# B&R Automation Studio project A2019059_Linka_Power_CP (part 29)

```iecst
        273:
            SC_P2_Srobovanie.StepName:='273 - Automaticky Rezim - model 5F, zasunutie skrutkovacky M4 a vypnutie prisavania skrutky';
            SC_P2_Srobovanie.IdleTime.PT:= T#200ms;
            SC_P2_Srobovanie.AlarmTime.PT:= T#5s;

            IF NOT SC_P2_Srobovanie.Switch1 THEN
                P2_Srobovanie.OUT.SkrutkM4_VYSUN_YV24:= FALSE;
                P2_Srobovanie.OUT.SkrutkM4_PrisavSkrutky_RUN_YV26:= FALSE;
                SC_P2_Srobovanie.Switch1:= TRUE;
            END_IF

            IF P2_Srobovanie.IN.SkrutkM4_ZASUNUTY_MS10 THEN
                SC_P2_Srobovanie.ResetStep:= TRUE;
                SC_P2_Srobovanie.Step:= 274;
            END_IF

        274:
            SC_P2_Srobovanie.StepName:='274 - Automaticky Rezim - model 5F, signal skrutka M4 odobrata';
            SC_P2_Srobovanie.IdleTime.PT:= T#200ms;
            SC_P2_Srobovanie.AlarmTime.PT:= T#5s;

            IF NOT SC_P2_Srobovanie.Switch1 THEN
                P2_Srobovanie.SkrutkovaciSet_M4.SkrutkaM4_Odobrata:= TRUE;
                SC_P2_Srobovanie.Switch1:= TRUE;
            END_IF

            IF NOT P2_Srobovanie.SkrutkovaciSet_M4.SkrutkaM4_Pripravena THEN
                P2_Srobovanie.SkrutkovaciSet_M4.SkrutkaM4_Odobrata:= FALSE;
                SC_P2_Srobovanie.ResetStep:= TRUE;
                SC_P2_Srobovanie.Step:= 275;
            END_IF

        275:
            SC_P2_Srobovanie.StepName:='275 - Automaticky Rezim - model 5F, kontrola vysledkov skrutkovania pravej skrutky M4';
            SC_P2_Srobovanie.IdleTime.PT:= T#200ms;
            SC_P2_Srobovanie.AlarmTime.PT:= T#5s;

            IF P2_Srobovanie.Skrutkovacka_M4.Stav_VysledokUtahovania_OK THEN
                P2_Srobovanie.STAV.Vysledok_Srobovania:= 'OK';
                P2_Srobovanie.OUT.KOM_Srobovanie_Ukoncene:= TRUE;
                SC_P2_Srobovanie.ResetStep:= TRUE;
                SC_P2_Srobovanie.Step:= 278;
            ELSIF P2_Srobovanie.Skrutkovacka_M4.Stav_VysledokUtahovania_NG THEN
                P2_Srobovanie.STAV.Vysledok_Srobovania:= 'NG';
                P2_Srobovanie.OUT.KOM_Srobovanie_Ukoncene:= TRUE;
                SC_P2_Srobovanie.ResetStep:= TRUE;
                SC_P2_Srobovanie.Step:= 278;
            END_IF

        278:
            SC_P2_Srobovanie.StepName:='278 - Automaticky Rezim - model 5F, cakam na zrusenie signalu zaskrutkuj pravu srobu M4';
            SC_P2_Srobovanie.IdleTime.PT:= T#200ms;
            SC_P2_Srobovanie.AlarmTime.PT:= T#5s;

            IF NOT P2_StoperSrobovania.OUT.KOM_5F_ZasrobujPravuSkrutkuM4 THEN
                P2_Srobovanie.OUT.KOM_Srobovanie_Ukoncene:= FALSE;
                SC_P2_Srobovanie.ResetStep:= TRUE;
                SC_P2_Srobovanie.Step:= 100;
            END_IF

            //**********************************************************************Model 5H*******************************************************************************************//
            //Zaskrutkovanie lavej skrutky M5//

        300:
            SC_P2_Srobovanie.StepName:='300 - Automaticky Rezim - model 5H, napolohovanie zadnej skrutkovacky M5 na poziciu lavej skrutky M5';
            SC_P2_Srobovanie.IdleTime.PT:= T#200ms;
            SC_P2_Srobovanie.AlarmTime.PT:= T#5s;

            P2_Robot.KOM_OUT.ManipSrobovania_BezpecnaPozicia:= FALSE;

            P2_Srobovanie.PAR.OsX_ZadanaPozicia:= P2_RemPremenne.P2_Srob5H_PozX_LavejSkrutkyM5; //mm
            P2_Srobovanie.PAR.OsY_ZadanaPozicia:= P2_RemPremenne.P2_Srob5H_PozY_LavejSkrutkyM5; //mm

            IF NOT SC_P2_Srobovanie.Switch1 AND SC_OvlManipulatora_OsX.Step = 1 AND SC_OvlManipulatora_OsY.Step = 1 AND P2_Srobovacky_VychodziaPozicia AND Safety.STAV.P2_ZonaBunky_AKTIVNA  THEN
                OsX_POLOHUJ:= TRUE;
                OsY_POLOHUJ:= TRUE;
                SC_P2_Srobovanie.Switch1:= TRUE;
            END_IF

            IF P2_Srobovanie.STAV.OsX_PoziciaDosiahnuta AND P2_Srobovanie.STAV.OsY_PoziciaDosiahnuta THEN
                P2_Srobovanie.STAV.OsX_PoziciaDosiahnuta:= FALSE;
                P2_Srobovanie.STAV.OsY_PoziciaDosiahnuta:= FALSE;
                IF P2_Srobovanie.RR_PolohujNaPoziciuSkrutky_5H THEN
                    P2_Srobovanie.RR_PolohujNaPoziciuSkrutky_5H:= FALSE;
                    P2_Srobovanie.RR_PolohujNaPoziciuSkrutky_4F:= FALSE;
                    P2_Srobovanie.RR_PolohujNaPoziciuSkrutky_5F:= FALSE;
                    SC_P2_Srobovanie.ResetStep:= TRUE;
                    SC_P2_Srobovanie.Step:= 700;
                ELSE
                    SC_P2_Srobovanie.ResetStep:= TRUE;
                    SC_P2_Srobovanie.Step:= 303;
                END_IF
            END_IF

        303:
            SC_P2_Srobovanie.StepName:='303 - Automaticky Rezim - model 5H, vymazanie vysledkov srobovania';
            SC_P2_Srobovanie.IdleTime.PT:= T#2s;
            SC_P2_Srobovanie.AlarmTime.PT:= T#5s;

            IF NOT SC_P2_Srobovanie.Switch1 THEN
                P2_Srobovanie.Skrutkovacka_M5.RESET_Vysledkov:= TRUE;
                SC_P2_Srobovanie.Switch1:= TRUE;
            END_IF

            IF NOT P2_Srobovanie.Skrutkovacka_M5.Stav_VysledokUtahovania_NG AND NOT P2_Srobovanie.Skrutkovacka_M5.Stav_VysledokUtahovania_OK AND NOT P2_Srobovanie.Skrutkovacka_M5.Stav_UtahovanieUkoncene THEN
                P2_Srobovanie.Skrutkovacka_M5.RESET_Vysledkov:= FALSE;
                SC_P2_Srobovanie.ResetStep:= TRUE;
                SC_P2_Srobovanie.Step:= 305;
            END_IF

        305:
            SC_P2_Srobovanie.StepName:='305 - Automaticky Rezim - model 5H, kontrola skrutky M5 v skrutkovacke';
            SC_P2_Srobovanie.IdleTime.PT:= T#5s;
            SC_P2_Srobovanie.AlarmTime.PT:= T#30s;
            SC_P2_Srobovanie.AlarmTime.IN:= TRUE;

            IF P2_Srobovanie.SkrutkovaciSet_M5.SkrutkaM5_Pripravena AND P2_Srobovanie.Skrutkovacka_M5.Stav_READY_to_START AND NOT PAUZA THEN
                SC_P2_Srobovanie.ResetStep:= TRUE;
                SC_P2_Srobovanie.Step:= 308;
            ELSIF SC_P2_Srobovanie.AlarmTime.Q THEN
                IF NOT P2_Srobovanie.SkrutkovaciSet_M5.SkrutkaM5_Pripravena THEN
                    P2_Alarmy[238]:= TRUE;
                END_IF
                IF NOT P2_Srobovanie.Skrutkovacka_M5.Stav_READY_to_START THEN
                    P2_Alarmy[276]:= TRUE;
                END_IF
                P2_StoperSrobovania.STAV.Porucha:= TRUE;
                P2_Srobovanie.OUT.KOM_Srobovanie_Ukoncene:= TRUE;
                SC_P2_Srobovanie.ResetStep:= TRUE;
                SC_P2_Srobovanie.Step:= 318;
            END_IF

        308:
            SC_P2_Srobovanie.StepName:='308 - Automaticky Rezim - model 5H, vysunutie skrutkovacky M5';
            SC_P2_Srobovanie.IdleTime.PT:= T#2s;
            SC_P2_Srobovanie.AlarmTime.PT:= T#5s;

            SC_P2_Srobovanie.AlarmTime.IN:= (P2_Srobovanie.IN.SkrutkM5_VysunutieHrotu_IOS5 < 2);

            IF NOT SC_P2_Srobovanie.Switch1 THEN
                P2_Srobovanie.OUT.SkrutkM5_PrisavSkrutky_RUN_YV16:= TRUE;
                P2_Srobovanie.OUT.SkrutkM5_VYSUN_YV14:= TRUE;
                P2_Srobovanie.Skrutkovacka_M5.START_Utahovania:= TRUE;
                SC_P2_Srobovanie.Switch1:= TRUE;
            END_IF

            IF NOT P2_Srobovanie.Skrutkovacka_M5.Stav_UtahovanieUkoncene AND P2_Srobovanie.IN.SkrutkM5_VysunutieHrotu_IOS5 > 2 AND NOT TEST THEN
                SC_P2_Srobovanie.ResetStep:= TRUE;
                SC_P2_Srobovanie.Step:= 310;
            ELSIF SC_P2_Srobovanie.AlarmTime.Q AND NOT TEST THEN
                P2_Alarmy[269]:= TRUE;
                P2_StoperSrobovania.STAV.Porucha:= TRUE;
                P2_Srobovanie.OUT.SkrutkM5_VYSUN_YV14:= FALSE;
                P2_Srobovanie.Skrutkovacka_M5.START_Utahovania:= FALSE;
                P2_Srobovanie.OUT.KOM_Srobovanie_Ukoncene:= TRUE;
                SC_P2_Srobovanie.ResetStep:= TRUE;
                SC_P2_Srobovanie.Step:= 318;
            END_IF

        310:
            SC_P2_Srobovanie.StepName:='310 - Automaticky Rezim - model 5H, cakam na ukoncenie skrutkovania skrutkovacky M5';
            SC_P2_Srobovanie.IdleTime.PT:= T#30s;
            SC_P2_Srobovanie.AlarmTime.PT:= T#10s;
            SC_P2_Srobovanie.IdleTime.IN:= TRUE;
            SC_P2_Srobovanie.AlarmTime.IN:= TRUE;

            IF P2_Srobovanie.Skrutkovacka_M5.Stav_UtahovanieUkoncene THEN
                P2_Srobovanie.Skrutkovacka_M5.START_Utahovania:= FALSE;
                CasSrobovania:= TIME_TO_REAL(SC_P2_Srobovanie.IdleTime.ET);
                Reports.Skrutkovacky.VyskaSkrutkovania.P2_LavaSkrutkaM5:= REAL_TO_STRING(P2_Srobovanie.IN.SkrutkM5_VysunutieHrotu_IOS5);
                Reports.Skrutkovacky.CasSkrutkovania.P2_LavaSkrutkaM5:= REAL_TO_STRING(CasSrobovania/1000);
                SC_P2_Srobovanie.ResetStep:= TRUE;
                SC_P2_Srobovanie.Step:= 313;
            ELSIF SC_P2_Srobovanie.AlarmTime.Q THEN
                P2_Alarmy[273]:= TRUE;
                P2_StoperSrobovania.STAV.Porucha:= TRUE;
                P2_Srobovanie.OUT.SkrutkM5_VYSUN_YV14:= FALSE;
                P2_Srobovanie.Skrutkovacka_M5.START_Utahovania:= FALSE;
                P2_Srobovanie.OUT.KOM_Srobovanie_Ukoncene:= TRUE;
                SC_P2_Srobovanie.ResetStep:= TRUE;
                SC_P2_Srobovanie.Step:= 318;
            END_IF

        313:
            SC_P2_Srobovanie.StepName:='313 - Automaticky Rezim - model 5H, zasunutie skrutkovacky M5 a vypnutie prisavania skrutky';
            SC_P2_Srobovanie.IdleTime.PT:= T#200ms;
            SC_P2_Srobovanie.AlarmTime.PT:= T#5s;

            IF NOT SC_P2_Srobovanie.Switch1 THEN
                P2_Srobovanie.OUT.SkrutkM5_VYSUN_YV14:= FALSE;
                P2_Srobovanie.OUT.SkrutkM5_PrisavSkrutky_RUN_YV16:= FALSE;
                SC_P2_Srobovanie.Switch1:= TRUE;
            END_IF

            IF P2_Srobovanie.IN.SkrutkM5_ZASUNUTY_MS11 THEN
                SC_P2_Srobovanie.ResetStep:= TRUE;
                SC_P2_Srobovanie.Step:= 314;
            END_IF

        314:
            SC_P2_Srobovanie.StepName:='314 - Automaticky Rezim - model 5H, signal skrutka M5 odobrata';
            SC_P2_Srobovanie.IdleTime.PT:= T#200ms;
            SC_P2_Srobovanie.AlarmTime.PT:= T#5s;

            IF NOT SC_P2_Srobovanie.Switch1 THEN
                P2_Srobovanie.SkrutkovaciSet_M5.SkrutkaM5_Odobrata:= TRUE;
                SC_P2_Srobovanie.Switch1:= TRUE;
            END_IF

            IF NOT P2_Srobovanie.SkrutkovaciSet_M5.SkrutkaM5_Pripravena THEN
                P2_Srobovanie.SkrutkovaciSet_M5.SkrutkaM5_Odobrata:= FALSE;
                SC_P2_Srobovanie.ResetStep:= TRUE;
                SC_P2_Srobovanie.Step:= 315;
            END_IF

        315:
            SC_P2_Srobovanie.StepName:='315 - Automaticky Rezim - model 5H, kontrola vysledkov skrutkovania lavej skrutky M5';
            SC_P2_Srobovanie.IdleTime.PT:= T#200ms;
            SC_P2_Srobovanie.AlarmTime.PT:= T#5s;

            IF P2_Srobovanie.Skrutkovacka_M5.Stav_VysledokUtahovania_OK THEN
                P2_Srobovanie.STAV.Vysledok_Srobovania:= 'OK';
                P2_Srobovanie.OUT.KOM_Srobovanie_Ukoncene:= TRUE;
                SC_P2_Srobovanie.ResetStep:= TRUE;
                SC_P2_Srobovanie.Step:= 318;
            ELSIF P2_Srobovanie.Skrutkovacka_M5.Stav_VysledokUtahovania_NG THEN
                P2_Srobovanie.STAV.Vysledok_Srobovania:= 'NG';
                P2_Srobovanie.OUT.KOM_Srobovanie_Ukoncene:= TRUE;
                SC_P2_Srobovanie.ResetStep:= TRUE;
                SC_P2_Srobovanie.Step:= 318;
            END_IF

        318:
            SC_P2_Srobovanie.StepName:='318 - Automaticky Rezim - model 5H, cakam na zrusenie signalu zaskrutkuj lavu srobu M5';
            SC_P2_Srobovanie.IdleTime.PT:= T#200ms;
            SC_P2_Srobovanie.AlarmTime.PT:= T#5s;

            IF NOT P2_StoperSrobovania.OUT.KOM_5H_ZasrobujLavuSkrutkuM5 THEN
                P2_Srobovanie.OUT.KOM_Srobovanie_Ukoncene:= FALSE;
                SC_P2_Srobovanie.ResetStep:= TRUE;
                SC_P2_Srobovanie.Step:= 100;
            END_IF

            //Zaskrutkovanie pravej skrutky M5//

        320:
            SC_P2_Srobovanie.StepName:='320 - Automaticky Rezim - model 5H, napolohovanie zadnej skrutkovacky M5 na poziciu pravej skrutky M5';
            SC_P2_Srobovanie.IdleTime.PT:= T#200ms;
            SC_P2_Srobovanie.AlarmTime.PT:= T#5s;

            P2_Robot.KOM_OUT.ManipSrobovania_BezpecnaPozicia:= FALSE;

            P2_Srobovanie.PAR.OsX_ZadanaPozicia:= P2_RemPremenne.P2_Srob5H_PozX_PravejSkrutkyM5; //mm
            P2_Srobovanie.PAR.OsY_ZadanaPozicia:= P2_RemPremenne.P2_Srob5H_PozY_PravejSkrutkyM5; //mm

            IF NOT SC_P2_Srobovanie.Switch1 AND SC_OvlManipulatora_OsX.Step = 1 AND SC_OvlManipulatora_OsY.Step = 1 AND P2_Srobovacky_VychodziaPozicia AND Safety.STAV.P2_ZonaBunky_AKTIVNA THEN
                OsX_POLOHUJ:= TRUE;
                OsY_POLOHUJ:= TRUE;
                SC_P2_Srobovanie.Switch1:= TRUE;
            END_IF

            IF P2_Srobovanie.STAV.OsX_PoziciaDosiahnuta AND P2_Srobovanie.STAV.OsY_PoziciaDosiahnuta THEN
                P2_Srobovanie.STAV.OsX_PoziciaDosiahnuta:= FALSE;
                P2_Srobovanie.STAV.OsY_PoziciaDosiahnuta:= FALSE;
                IF P2_Srobovanie.RR_PolohujNaPoziciuSkrutky_5H THEN
                    P2_Srobovanie.RR_PolohujNaPoziciuSkrutky_5H:= FALSE;
                    P2_Srobovanie.RR_PolohujNaPoziciuSkrutky_4F:= FALSE;
                    P2_Srobovanie.RR_PolohujNaPoziciuSkrutky_5F:= FALSE;
                    SC_P2_Srobovanie.ResetStep:= TRUE;
                    SC_P2_Srobovanie.Step:= 700;
                ELSE
                    SC_P2_Srobovanie.ResetStep:= TRUE;
                    SC_P2_Srobovanie.Step:= 323;
                END_IF
            END_IF

        323:
            SC_P2_Srobovanie.StepName:='323 - Automaticky Rezim - model 5H, vymazanie vysledkov srobovania';
            SC_P2_Srobovanie.IdleTime.PT:= T#2s;
            SC_P2_Srobovanie.AlarmTime.PT:= T#5s;

            IF NOT SC_P2_Srobovanie.Switch1 THEN
                P2_Srobovanie.Skrutkovacka_M5.RESET_Vysledkov:= TRUE;
                SC_P2_Srobovanie.Switch1:= TRUE;
            END_IF

            IF NOT P2_Srobovanie.Skrutkovacka_M5.Stav_VysledokUtahovania_NG AND NOT P2_Srobovanie.Skrutkovacka_M5.Stav_VysledokUtahovania_OK AND NOT P2_Srobovanie.Skrutkovacka_M5.Stav_UtahovanieUkoncene THEN
                P2_Srobovanie.Skrutkovacka_M5.RESET_Vysledkov:= FALSE;
                SC_P2_Srobovanie.ResetStep:= TRUE;
                SC_P2_Srobovanie.Step:= 325;
            END_IF

        325:
            SC_P2_Srobovanie.StepName:='325 - Automaticky Rezim - model 5H, kontrola skrutky M5 v skrutkovacke';
            SC_P2_Srobovanie.IdleTime.PT:= T#5s;
            SC_P2_Srobovanie.AlarmTime.PT:= T#30s;
            SC_P2_Srobovanie.AlarmTime.IN:= TRUE;

            IF P2_Srobovanie.SkrutkovaciSet_M5.SkrutkaM5_Pripravena AND P2_Srobovanie.Skrutkovacka_M5.Stav_READY_to_START AND NOT PAUZA THEN
                SC_P2_Srobovanie.ResetStep:= TRUE;
                SC_P2_Srobovanie.Step:= 328;
            ELSIF SC_P2_Srobovanie.AlarmTime.Q THEN
                IF NOT P2_Srobovanie.SkrutkovaciSet_M5.SkrutkaM5_Pripravena THEN
                    P2_Alarmy[238]:= TRUE;
                END_IF
                IF NOT P2_Srobovanie.Skrutkovacka_M5.Stav_READY_to_START THEN
                    P2_Alarmy[276]:= TRUE;
                END_IF
                P2_StoperSrobovania.STAV.Porucha:= TRUE;
                P2_Srobovanie.OUT.KOM_Srobovanie_Ukoncene:= TRUE;
                SC_P2_Srobovanie.ResetStep:= TRUE;
                SC_P2_Srobovanie.Step:= 338;
            END_IF

        328:
            SC_P2_Srobovanie.StepName:='328 - Automaticky Rezim - model 5H, vysunutie skrutkovacky M5';
            SC_P2_Srobovanie.IdleTime.PT:= T#2s;
            SC_P2_Srobovanie.AlarmTime.PT:= T#5s;

            SC_P2_Srobovanie.AlarmTime.IN:= (P2_Srobovanie.IN.SkrutkM5_VysunutieHrotu_IOS5 < 2);

            IF NOT SC_P2_Srobovanie.Switch1 THEN
                P2_Srobovanie.OUT.SkrutkM5_PrisavSkrutky_RUN_YV16:= TRUE;
                P2_Srobovanie.OUT.SkrutkM5_VYSUN_YV14:= TRUE;
                P2_Srobovanie.Skrutkovacka_M5.START_Utahovania:= TRUE;
                SC_P2_Srobovanie.Switch1:= TRUE;
            END_IF

            IF NOT P2_Srobovanie.Skrutkovacka_M5.Stav_UtahovanieUkoncene AND P2_Srobovanie.IN.SkrutkM5_VysunutieHrotu_IOS5 > 2 THEN
                SC_P2_Srobovanie.ResetStep:= TRUE;
                SC_P2_Srobovanie.Step:= 330;
            ELSIF SC_P2_Srobovanie.AlarmTime.Q THEN
                P2_Alarmy[269]:= TRUE;
                P2_StoperSrobovania.STAV.Porucha:= TRUE;
                P2_Srobovanie.OUT.SkrutkM5_VYSUN_YV14:= FALSE;
                P2_Srobovanie.Skrutkovacka_M5.START_Utahovania:= FALSE;
                P2_Srobovanie.OUT.KOM_Srobovanie_Ukoncene:= TRUE;
                SC_P2_Srobovanie.ResetStep:= TRUE;
                SC_P2_Srobovanie.Step:= 338;
            END_IF

        330:
            SC_P2_Srobovanie.StepName:='330 - Automaticky Rezim - model 5H, cakam na ukoncenie skrutkovania skrutkovacky M5';
            SC_P2_Srobovanie.IdleTime.PT:= T#30s;
            SC_P2_Srobovanie.AlarmTime.PT:= T#10s;
            SC_P2_Srobovanie.IdleTime.IN:= TRUE;
            SC_P2_Srobovanie.AlarmTime.IN:= TRUE;

            IF P2_Srobovanie.Skrutkovacka_M5.Stav_UtahovanieUkoncene AND NOT P2_Robot.KOM_IN.Stav_BusbaryUvolnene THEN
                P2_Srobovanie.Skrutkovacka_M5.START_Utahovania:= FALSE;
                CasSrobovania:= TIME_TO_REAL(SC_P2_Srobovanie.IdleTime.ET);
                Reports.Skrutkovacky.VyskaSkrutkovania.P2_PravaSkrutkaM5:= REAL_TO_STRING(P2_Srobovanie.IN.SkrutkM5_VysunutieHrotu_IOS5);
                Reports.Skrutkovacky.CasSkrutkovania.P2_PravaSkrutkaM5:= REAL_TO_STRING(CasSrobovania/1000);
                SC_P2_Srobovanie.ResetStep:= TRUE;
                SC_P2_Srobovanie.Step:= 332;
            ELSIF SC_P2_Srobovanie.AlarmTime.Q THEN
                P2_Alarmy[273]:= TRUE;
                P2_StoperSrobovania.STAV.Porucha:= TRUE;
                P2_Srobovanie.OUT.SkrutkM5_VYSUN_YV14:= FALSE;
                P2_Srobovanie.Skrutkovacka_M5.START_Utahovania:= FALSE;
                P2_Srobovanie.OUT.KOM_Srobovanie_Ukoncene:= TRUE;
                SC_P2_Srobovanie.ResetStep:= TRUE;
                SC_P2_Srobovanie.Step:= 338;
            END_IF

        332:
            SC_P2_Srobovanie.StepName:='332 - Automaticky Rezim - model 5H, uvolnenie busbarov';
            SC_P2_Srobovanie.IdleTime.PT:= T#30s;
            SC_P2_Srobovanie.AlarmTime.PT:= T#5s;

            IF NOT SC_P2_Srobovanie.Switch1 THEN
                P2_Robot.KOM_OUT.UvolniBusbary:= TRUE;
                SC_P2_Srobovanie.Switch1:= TRUE;
            END_IF

            IF P2_Robot.KOM_IN.Stav_BusbaryUvolnene THEN
                P2_Robot.KOM_OUT.UvolniBusbary:= FALSE;
                SC_P2_Srobovanie.ResetStep:= TRUE;
                SC_P2_Srobovanie.Step:= 333;
            END_IF

        333:
            SC_P2_Srobovanie.StepName:='333 - Automaticky Rezim - model 5H, zasunutie skrutkovacky M5 a vypnutie prisavania skrutky';
            SC_P2_Srobovanie.IdleTime.PT:= T#200ms;
            SC_P2_Srobovanie.AlarmTime.PT:= T#5s;

            IF NOT SC_P2_Srobovanie.Switch1 THEN
                P2_Srobovanie.OUT.SkrutkM5_VYSUN_YV14:= FALSE;
                P2_Srobovanie.OUT.SkrutkM5_PrisavSkrutky_RUN_YV16:= FALSE;
                SC_P2_Srobovanie.Switch1:= TRUE;
            END_IF

            IF P2_Srobovanie.IN.SkrutkM5_ZASUNUTY_MS11 THEN
                SC_P2_Srobovanie.ResetStep:= TRUE;
                SC_P2_Srobovanie.Step:= 334;
            END_IF

        334:
            SC_P2_Srobovanie.StepName:='334 - Automaticky Rezim - model 5H, signal skrutka M5 odobrata';
            SC_P2_Srobovanie.IdleTime.PT:= T#200ms;
            SC_P2_Srobovanie.AlarmTime.PT:= T#5s;

            IF NOT SC_P2_Srobovanie.Switch1 THEN
                P2_Srobovanie.SkrutkovaciSet_M5.SkrutkaM5_Odobrata:= TRUE;
                SC_P2_Srobovanie.Switch1:= TRUE;
            END_IF

            IF NOT P2_Srobovanie.SkrutkovaciSet_M5.SkrutkaM5_Pripravena THEN
                P2_Srobovanie.SkrutkovaciSet_M5.SkrutkaM5_Odobrata:= FALSE;
                SC_P2_Srobovanie.ResetStep:= TRUE;
                SC_P2_Srobovanie.Step:= 335;
            END_IF

        335:
            SC_P2_Srobovanie.StepName:='335 - Automaticky Rezim - model 5H, kontrola vysledkov skrutkovania pravej skrutky M5';
            SC_P2_Srobovanie.IdleTime.PT:= T#200ms;
            SC_P2_Srobovanie.AlarmTime.PT:= T#5s;

            IF P2_Srobovanie.Skrutkovacka_M5.Stav_VysledokUtahovania_OK THEN
                P2_Srobovanie.STAV.Vysledok_Srobovania:= 'OK';
                P2_Srobovanie.OUT.KOM_Srobovanie_Ukoncene:= TRUE;
                SC_P2_Srobovanie.ResetStep:= TRUE;
                SC_P2_Srobovanie.Step:= 338;
            ELSIF P2_Srobovanie.Skrutkovacka_M5.Stav_VysledokUtahovania_NG THEN
                P2_Srobovanie.STAV.Vysledok_Srobovania:= 'NG';
                P2_Srobovanie.OUT.KOM_Srobovanie_Ukoncene:= TRUE;
                SC_P2_Srobovanie.ResetStep:= TRUE;
                SC_P2_Srobovanie.Step:= 338;
            END_IF

        338:
            SC_P2_Srobovanie.StepName:='338 - Automaticky Rezim - model 5H, cakam na zrusenie signalu zaskrutkuj pravu srobu M5';
            SC_P2_Srobovanie.IdleTime.PT:= T#200ms;
            SC_P2_Srobovanie.AlarmTime.PT:= T#5s;

            IF NOT P2_StoperSrobovania.OUT.KOM_5H_ZasrobujPravuSkrutkuM5 THEN
                P2_Srobovanie.OUT.KOM_Srobovanie_Ukoncene:= FALSE;
                SC_P2_Srobovanie.ResetStep:= TRUE;
                SC_P2_Srobovanie.Step:= 100;
            END_IF

            //Zaskrutkovanie skrutky M4//

        340:
            SC_P2_Srobovanie.StepName:='340 - Automaticky Rezim - model 5H, napolohovanie strednej skrutkovacky M4 na poziciu skrutky M4';
            SC_P2_Srobovanie.IdleTime.PT:= T#200ms;
            SC_P2_Srobovanie.AlarmTime.PT:= T#5s;

            P2_Robot.KOM_OUT.ManipSrobovania_BezpecnaPozicia:= FALSE;

            P2_Srobovanie.PAR.OsX_ZadanaPozicia:= P2_RemPremenne.P2_Srob5H_PozX_SkrutkyM4; //mm
            P2_Srobovanie.PAR.OsY_ZadanaPozicia:= P2_RemPremenne.P2_Srob5H_PozY_SkrutkyM4; //mm

            IF NOT SC_P2_Srobovanie.Switch1 AND SC_OvlManipulatora_OsX.Step = 1 AND SC_OvlManipulatora_OsY.Step = 1 AND P2_Srobovacky_VychodziaPozicia AND Safety.STAV.P2_ZonaBunky_AKTIVNA THEN
                OsX_POLOHUJ:= TRUE;
                OsY_POLOHUJ:= TRUE;
                SC_P2_Srobovanie.Switch1:= TRUE;
            END_IF

            IF P2_Srobovanie.STAV.OsX_PoziciaDosiahnuta AND P2_Srobovanie.STAV.OsY_PoziciaDosiahnuta THEN
                P2_Srobovanie.STAV.OsX_PoziciaDosiahnuta:= FALSE;
                P2_Srobovanie.STAV.OsY_PoziciaDosiahnuta:= FALSE;
                IF P2_Srobovanie.RR_PolohujNaPoziciuSkrutky_5H THEN
                    P2_Srobovanie.RR_PolohujNaPoziciuSkrutky_5H:= FALSE;
                    P2_Srobovanie.RR_PolohujNaPoziciuSkrutky_4F:= FALSE;
                    P2_Srobovanie.RR_PolohujNaPoziciuSkrutky_5F:= FALSE;
                    SC_P2_Srobovanie.ResetStep:= TRUE;
                    SC_P2_Srobovanie.Step:= 700;
                ELSE
                    SC_P2_Srobovanie.ResetStep:= TRUE;
                    SC_P2_Srobovanie.Step:= 343;
                END_IF
            END_IF

        343:
            SC_P2_Srobovanie.StepName:='343 - Automaticky Rezim - model 5H, vymazanie vysledkov srobovania';
            SC_P2_Srobovanie.IdleTime.PT:= T#2s;
            SC_P2_Srobovanie.AlarmTime.PT:= T#5s;

            IF NOT SC_P2_Srobovanie.Switch1 THEN
                P2_Srobovanie.Skrutkovacka_M4.RESET_Vysledkov:= TRUE;
                SC_P2_Srobovanie.Switch1:= TRUE;
            END_IF

            IF NOT P2_Srobovanie.Skrutkovacka_M4.Stav_VysledokUtahovania_NG AND NOT P2_Srobovanie.Skrutkovacka_M4.Stav_VysledokUtahovania_OK AND NOT P2_Srobovanie.Skrutkovacka_M4.Stav_UtahovanieUkoncene THEN
                P2_Srobovanie.Skrutkovacka_M4.RESET_Vysledkov:= FALSE;
                SC_P2_Srobovanie.ResetStep:= TRUE;
                SC_P2_Srobovanie.Step:= 345;
            END_IF

        345:
            SC_P2_Srobovanie.StepName:='345 - Automaticky Rezim - model 5H, kontrola skrutky M4 v skrutkovacke';
            SC_P2_Srobovanie.IdleTime.PT:= T#5s;
            SC_P2_Srobovanie.AlarmTime.PT:= T#30s;
            SC_P2_Srobovanie.AlarmTime.IN:= TRUE;

            IF P2_Srobovanie.SkrutkovaciSet_M4.SkrutkaM4_Pripravena AND P2_Srobovanie.Skrutkovacka_M4.Stav_READY_to_START AND NOT PAUZA THEN
                SC_P2_Srobovanie.ResetStep:= TRUE;
                SC_P2_Srobovanie.Step:= 348;
            ELSIF SC_P2_Srobovanie.AlarmTime.Q THEN
                IF NOT P2_Srobovanie.SkrutkovaciSet_M4.SkrutkaM4_Pripravena THEN
                    P2_Alarmy[237]:= TRUE;
                END_IF
                IF NOT P2_Srobovanie.Skrutkovacka_M4.Stav_READY_to_START THEN
                    P2_Alarmy[275]:= TRUE;
                END_IF
                P2_StoperSrobovania.STAV.Porucha:= TRUE;
                P2_Srobovanie.OUT.KOM_Srobovanie_Ukoncene:= TRUE;
                SC_P2_Srobovanie.ResetStep:= TRUE;
                SC_P2_Srobovanie.Step:= 358;
            END_IF

        348:
            SC_P2_Srobovanie.StepName:='348 - Automaticky Rezim - model 5H, vysunutie skrutkovacky M4';
            SC_P2_Srobovanie.IdleTime.PT:= T#2s;
            SC_P2_Srobovanie.AlarmTime.PT:= T#5s;
            SC_P2_Srobovanie.IdleTime.IN:= TRUE;

            SC_P2_Srobovanie.AlarmTime.IN:= (P2_Srobovanie.IN.SkrutkM4_VysunutieHrotu_IOS4 < 2);

            IF NOT SC_P2_Srobovanie.Switch1 THEN
                P2_Srobovanie.OUT.SkrutkM4_VYSUN_YV24:= TRUE;
                P2_Srobovanie.OUT.SkrutkM4_PrisavSkrutky_RUN_YV26:= TRUE;
                P2_Srobovanie.Skrutkovacka_M4.START_Utahovania:= TRUE;
                SC_P2_Srobovanie.Switch1:= TRUE;
            END_IF

            IF NOT P2_Srobovanie.Skrutkovacka_M4.Stav_UtahovanieUkoncene AND P2_Srobovanie.IN.SkrutkM4_VysunutieHrotu_IOS4 > 2 AND NOT TEST THEN
                SC_P2_Srobovanie.ResetStep:= TRUE;
                SC_P2_Srobovanie.Step:= 350;
            ELSIF SC_P2_Srobovanie.AlarmTime.Q AND NOT TEST THEN
                P2_Alarmy[268]:= TRUE;
                P2_StoperSrobovania.STAV.Porucha:= TRUE;
                P2_Srobovanie.OUT.SkrutkM4_PrisavSkrutky_RUN_YV26:= FALSE;
                P2_Srobovanie.Skrutkovacka_M4.START_Utahovania:= FALSE;
                P2_Srobovanie.OUT.KOM_Srobovanie_Ukoncene:= TRUE;
                SC_P2_Srobovanie.ResetStep:= TRUE;
                SC_P2_Srobovanie.Step:= 358;
            END_IF

        350:
            SC_P2_Srobovanie.StepName:='350 - Automaticky Rezim - model 5H, cakam na ukoncenie skrutkovania skrutkovacky M4';
            SC_P2_Srobovanie.IdleTime.PT:= T#30s;
            SC_P2_Srobovanie.AlarmTime.PT:= T#10s;
            SC_P2_Srobovanie.IdleTime.IN:= TRUE;
            SC_P2_Srobovanie.AlarmTime.IN:= TRUE;

            IF P2_Srobovanie.Skrutkovacka_M4.Stav_UtahovanieUkoncene THEN
                P2_Srobovanie.Skrutkovacka_M4.START_Utahovania:= FALSE;
                CasSrobovania:= TIME_TO_REAL(SC_P2_Srobovanie.IdleTime.ET);
                Reports.Skrutkovacky.VyskaSkrutkovania.P2_StrednaSkrutkaM4:= REAL_TO_STRING(P2_Srobovanie.IN.SkrutkM4_VysunutieHrotu_IOS4);
                Reports.Skrutkovacky.CasSkrutkovania.P2_StrednaSkrutkaM4:= REAL_TO_STRING(CasSrobovania/1000);
                SC_P2_Srobovanie.ResetStep:= TRUE;
                SC_P2_Srobovanie.Step:= 353;
            ELSIF SC_P2_Srobovanie.AlarmTime.Q THEN
                P2_Alarmy[272]:= TRUE;
                P2_StoperSrobovania.STAV.Porucha:= TRUE;
                P2_Srobovanie.OUT.SkrutkM4_PrisavSkrutky_RUN_YV26:= FALSE;
                P2_Srobovanie.Skrutkovacka_M4.START_Utahovania:= FALSE;
                P2_Srobovanie.OUT.KOM_Srobovanie_Ukoncene:= TRUE;
                SC_P2_Srobovanie.ResetStep:= TRUE;
                SC_P2_Srobovanie.Step:= 358;
            END_IF

        353:
            SC_P2_Srobovanie.StepName:='353 - Automaticky Rezim - model 5H, zasunutie skrutkovacky M4 a vypnutie prisavania skrutky';
            SC_P2_Srobovanie.IdleTime.PT:= T#200ms;
            SC_P2_Srobovanie.AlarmTime.PT:= T#5s;

            IF NOT SC_P2_Srobovanie.Switch1 THEN
                P2_Srobovanie.OUT.SkrutkM4_VYSUN_YV24:= FALSE;
                P2_Srobovanie.OUT.SkrutkM4_PrisavSkrutky_RUN_YV26:= FALSE;
                SC_P2_Srobovanie.Switch1:= TRUE;
            END_IF

            IF P2_Srobovanie.IN.SkrutkM4_ZASUNUTY_MS10 THEN
                SC_P2_Srobovanie.ResetStep:= TRUE;
                SC_P2_Srobovanie.Step:= 354;
            END_IF

        354:
            SC_P2_Srobovanie.StepName:='354 - Automaticky Rezim - model 5H, signal skrutka M4 odobrata';
            SC_P2_Srobovanie.IdleTime.PT:= T#200ms;
            SC_P2_Srobovanie.AlarmTime.PT:= T#5s;

            IF NOT SC_P2_Srobovanie.Switch1 THEN
                P2_Srobovanie.SkrutkovaciSet_M4.SkrutkaM4_Odobrata:= TRUE;
                SC_P2_Srobovanie.Switch1:= TRUE;
            END_IF

            IF NOT P2_Srobovanie.SkrutkovaciSet_M4.SkrutkaM4_Pripravena THEN
                P2_Srobovanie.SkrutkovaciSet_M4.SkrutkaM4_Odobrata:= FALSE;
                SC_P2_Srobovanie.ResetStep:= TRUE;
                SC_P2_Srobovanie.Step:= 355;
            END_IF

        355:
            SC_P2_Srobovanie.StepName:='355 - Automaticky Rezim - model 5H, kontrola vysledkov skrutkovania skrutky M4';
            SC_P2_Srobovanie.IdleTime.PT:= T#200ms;
            SC_P2_Srobovanie.AlarmTime.PT:= T#5s;

            IF P2_Srobovanie.Skrutkovacka_M4.Stav_VysledokUtahovania_OK THEN
                P2_Srobovanie.STAV.Vysledok_Srobovania:= 'OK';
                P2_Srobovanie.OUT.KOM_Srobovanie_Ukoncene:= TRUE;
                SC_P2_Srobovanie.ResetStep:= TRUE;
                SC_P2_Srobovanie.Step:= 358;
            ELSIF P2_Srobovanie.Skrutkovacka_M4.Stav_VysledokUtahovania_NG THEN
                P2_Srobovanie.STAV.Vysledok_Srobovania:= 'NG';
                P2_Srobovanie.OUT.KOM_Srobovanie_Ukoncene:= TRUE;
                SC_P2_Srobovanie.ResetStep:= TRUE;
                SC_P2_Srobovanie.Step:= 358;
            END_IF

        358:
            SC_P2_Srobovanie.StepName:='358 - Automaticky Rezim - model 5H, cakam na zrusenie signalu zaskrutkuj srobu M4';
            SC_P2_Srobovanie.IdleTime.PT:= T#200ms;
            SC_P2_Srobovanie.AlarmTime.PT:= T#5s;

            IF NOT P2_StoperSrobovania.OUT.KOM_5H_ZasrobujSkrutkuM4 THEN
                P2_Srobovanie.OUT.KOM_Srobovanie_Ukoncene:= FALSE;
                SC_P2_Srobovanie.ResetStep:= TRUE;
                SC_P2_Srobovanie.Step:= 100;
            END_IF

            //Presun manipulátora do pozície VPRED//

        400:
            SC_P2_Srobovanie.StepName:='400 - Automaticky Rezim - napolohovanie manipulatora do prednej pozicie';
            SC_P2_Srobovanie.IdleTime.PT:= T#200ms;
            SC_P2_Srobovanie.AlarmTime.PT:= T#5s;

            (*P2_Robot.KOM_OUT.ManipSrobovania_BezpecnaPozicia:= FALSE;*)

            P2_Srobovanie.PAR.OsX_ZadanaPozicia:= 0; //mm
            P2_Srobovanie.PAR.OsY_ZadanaPozicia:= 320; //mm

            IF NOT SC_P2_Srobovanie.Switch1 AND SC_OvlManipulatora_OsX.Step = 1 AND SC_OvlManipulatora_OsY.Step = 1 AND P2_Srobovacky_VychodziaPozicia AND Safety.STAV.P2_ZonaBunky_AKTIVNA THEN
                OsX_POLOHUJ:= TRUE;
                OsY_POLOHUJ:= TRUE;
                SC_P2_Srobovanie.Switch1:= TRUE;
            END_IF

            IF P2_Srobovanie.STAV.OsX_PoziciaDosiahnuta AND P2_Srobovanie.STAV.OsY_PoziciaDosiahnuta THEN
                P2_Srobovanie.STAV.OsX_PoziciaDosiahnuta:= FALSE;
                P2_Srobovanie.STAV.OsY_PoziciaDosiahnuta:= FALSE;
                P2_Srobovanie.OUT.KOM_PresunVPRED_Ukonceny:= TRUE;
                SC_P2_Srobovanie.ResetStep:= TRUE;
                SC_P2_Srobovanie.Step:= 402;
            END_IF

        402:
            SC_P2_Srobovanie.StepName:='402 - Automaticky Rezim - cakam na zrusenie signalu presun manipulatora do prednej pozicie';
            SC_P2_Srobovanie.IdleTime.PT:= T#200ms;
            SC_P2_Srobovanie.AlarmTime.PT:= T#5s;

            IF NOT P2_StoperSrobovania.OUT.KOM_PresunManipulator_DOPREDU THEN
                SC_P2_Srobovanie.ResetStep:= TRUE;
                SC_P2_Srobovanie.Step:= 100;
            END_IF

            //Presun manipulatora do pozicie VZAD//

        420:
            SC_P2_Srobovanie.StepName:='420 - Automaticky Rezim - napolohovanie manipulatora do zadnej pozicie';
            SC_P2_Srobovanie.IdleTime.PT:= T#200ms;
            SC_P2_Srobovanie.AlarmTime.PT:= T#5s;

            P2_Robot.KOM_OUT.ManipSrobovania_BezpecnaPozicia:= FALSE;

            P2_Srobovanie.PAR.OsX_ZadanaPozicia:= 0; //mm
            P2_Srobovanie.PAR.OsY_ZadanaPozicia:= 0; //mm

            IF NOT SC_P2_Srobovanie.Switch1 AND SC_OvlManipulatora_OsX.Step = 1 AND SC_OvlManipulatora_OsY.Step = 1 AND P2_Srobovacky_VychodziaPozicia AND Safety.STAV.P2_ZonaBunky_AKTIVNA THEN
                OsX_POLOHUJ:= TRUE;
                OsY_POLOHUJ:= TRUE;
                SC_P2_Srobovanie.Switch1:= TRUE;
            END_IF

            IF P2_Srobovanie.STAV.OsX_PoziciaDosiahnuta AND P2_Srobovanie.STAV.OsY_PoziciaDosiahnuta THEN
                P2_Srobovanie.STAV.OsX_PoziciaDosiahnuta:= FALSE;
                P2_Srobovanie.STAV.OsY_PoziciaDosiahnuta:= FALSE;
                P2_Srobovanie.OUT.KOM_PresunVZAD_Ukonceny:= TRUE;
                SC_P2_Srobovanie.ResetStep:= TRUE;
                SC_P2_Srobovanie.Step:= 422;
            END_IF

        422:
            SC_P2_Srobovanie.StepName:='422 - Automaticky Rezim - cakam na zrusenie signalu presun manipulatora do zadnej pozicie';
            SC_P2_Srobovanie.IdleTime.PT:= T#200ms;
            SC_P2_Srobovanie.AlarmTime.PT:= T#5s;

            IF NOT P2_StoperSrobovania.OUT.KOM_PresunManipulator_DOZADU THEN
                SC_P2_Srobovanie.ResetStep:= TRUE;
                SC_P2_Srobovanie.Step:= 100;
            END_IF

            //***********************************************************Čistenie skrutkovačiek**********************************************************************//

            //Čistenie skrutkovačky M4//
        500:
            SC_P2_Srobovanie.StepName:='500 - Automaticky Rezim - cistenie skrutkovacky M4';
            SC_P2_Srobovanie.IdleTime.PT:= T#200ms;
            SC_P2_Srobovanie.AlarmTime.PT:= T#5s;

            P2_Srobovanie.PAR.OsX_ZadanaPozicia:= 50; //mm
            P2_Srobovanie.PAR.OsY_ZadanaPozicia:= 60; //mm

            IF NOT SC_P2_Srobovanie.Switch1 AND SC_OvlManipulatora_OsX.Step = 1 AND SC_OvlManipulatora_OsY.Step = 1 AND P2_Srobovacky_VychodziaPozicia AND Safety.STAV.P2_ZonaBunky_AKTIVNA THEN
                P2_Srobovanie.SkrutkovaciSet_M4.SkrutkaM4_Odobrata:= FALSE;
                P2_Srobovanie.SkrutkovaciSet_M4.Automat:= TRUE;
                P2_Srobovanie.SkrutkovaciSet_M4.Reset:= TRUE;
                OsX_POLOHUJ:= TRUE;
                SC_P2_Srobovanie.Switch1:= TRUE;
            END_IF

            IF NOT SC_P2_Srobovanie.Switch2 AND SC_OvlManipulatora_OsY.Step = 1 AND P2_Srobovacky_VychodziaPozicia AND P2_Srobovanie.STAV.OsX_PoziciaDosiahnuta AND Safety.STAV.P2_ZonaBunky_AKTIVNA THEN
                OsY_POLOHUJ:= TRUE;
                SC_P2_Srobovanie.Switch2:= TRUE;
            END_IF

            IF P2_Srobovanie.STAV.OsX_PoziciaDosiahnuta AND P2_Srobovanie.STAV.OsY_PoziciaDosiahnuta THEN
                P2_Srobovanie.STAV.OsX_PoziciaDosiahnuta:= FALSE;
                P2_Srobovanie.STAV.OsY_PoziciaDosiahnuta:= FALSE;
                SC_P2_Srobovanie.ResetStep:= TRUE;
                SC_P2_Srobovanie.Step:= 503;
            END_IF

        503:
            SC_P2_Srobovanie.StepName:='503 - Inicializacia - zahodenie skrutky M4';
            SC_P2_Srobovanie.IdleTime.PT:= T#30s;
            SC_P2_Srobovanie.AlarmTime.PT:= T#30s;
            SC_P2_Srobovanie.IdleTime.IN:= TRUE;

            IF NOT SC_P2_Srobovanie.Switch1 THEN
                P2_Srobovanie.SkrutkovaciSet_M4.Cistenie:= TRUE;
                SC_P2_Srobovanie.Switch1:= TRUE;
            END_IF

            IF P2_Srobovanie.SkrutkovaciSet_M4.CistenieUkoncene AND P2_Srobovanie.IN.SkrutkM4_ZASUNUTY_MS10 THEN
                P2_Srobovanie.SkrutkovaciSet_M4.Cistenie:= FALSE;
            END_IF

            IF NOT P2_Srobovanie.SkrutkovaciSet_M4.Cistenie AND P2_Srobovanie.SkrutkovaciSet_M4.SkrutkaM4_Pripravena AND SC_P2_Srobovanie.Switch1 THEN
                P2_Srobovanie.STAV.Cistenie_M4_BUSY:= FALSE;
                SC_P2_Srobovanie.ResetStep:= TRUE;
                SC_P2_Srobovanie.Step:= FazaNavratu;
            ELSIF SC_P2_Srobovanie.IdleTime.Q THEN
                SC_P2_Srobovanie.ResetStep:= TRUE;
                SC_P2_Srobovanie.Step:= 505;
            END_IF

        505:
            SC_P2_Srobovanie.StepName:='505 - Inicializacia - cakam na opatovne spustenie cistenia skrutkovacky M4';
            SC_P2_Srobovanie.IdleTime.PT:= T#2s;
            SC_P2_Srobovanie.AlarmTime.PT:= T#30s;

            IF NOT SC_P2_Srobovanie.Switch1 THEN
                P2_Srobovanie.SkrutkovaciSet_M4.Reset:= TRUE;
                P2_Srobovanie.SkrutkovaciSet_M4.Cistenie:= FALSE;
                SC_P2_Srobovanie.IdleTime.IN:= TRUE;
                SC_P2_Srobovanie.Switch1:= TRUE;
            END_IF

            IF SC_P2_Srobovanie.IdleTime.Q THEN
                SC_P2_Srobovanie.ResetStep:= TRUE;
                SC_P2_Srobovanie.Step:= 503;
            END_IF

            //Čistenie skrutkovačky M5//
        510:
            SC_P2_Srobovanie.StepName:='500 - Automaticky Rezim - cistenie skrutkovacky M5';
            SC_P2_Srobovanie.IdleTime.PT:= T#200ms;
            SC_P2_Srobovanie.AlarmTime.PT:= T#5s;

            P2_Srobovanie.PAR.OsX_ZadanaPozicia:= 50; //mm
            P2_Srobovanie.PAR.OsY_ZadanaPozicia:= 140; //mm

            IF NOT SC_P2_Srobovanie.Switch1 AND SC_OvlManipulatora_OsX.Step = 1 AND SC_OvlManipulatora_OsY.Step = 1 AND P2_Srobovacky_VychodziaPozicia AND Safety.STAV.P2_ZonaBunky_AKTIVNA THEN
                P2_Srobovanie.SkrutkovaciSet_M5.SkrutkaM5_Odobrata:= FALSE;
                P2_Srobovanie.SkrutkovaciSet_M5.Automat:= TRUE;
                P2_Srobovanie.SkrutkovaciSet_M5.Reset:= TRUE;
                OsX_POLOHUJ:= TRUE;
                SC_P2_Srobovanie.Switch1:= TRUE;
            END_IF

            IF NOT SC_P2_Srobovanie.Switch2 AND SC_OvlManipulatora_OsY.Step = 1 AND P2_Srobovacky_VychodziaPozicia AND P2_Srobovanie.STAV.OsX_PoziciaDosiahnuta AND Safety.STAV.P2_ZonaBunky_AKTIVNA THEN
                OsY_POLOHUJ:= TRUE;
                SC_P2_Srobovanie.Switch2:= TRUE;
            END_IF

            IF P2_Srobovanie.STAV.OsX_PoziciaDosiahnuta AND P2_Srobovanie.STAV.OsY_PoziciaDosiahnuta THEN
                P2_Srobovanie.STAV.OsX_PoziciaDosiahnuta:= FALSE;
                P2_Srobovanie.STAV.OsY_PoziciaDosiahnuta:= FALSE;
                SC_P2_Srobovanie.ResetStep:= TRUE;
                SC_P2_Srobovanie.Step:= 513;
            END_IF

        513:
            SC_P2_Srobovanie.StepName:='513 - Inicializacia - zahodenie skrutky M5';
            SC_P2_Srobovanie.IdleTime.PT:= T#30s;
            SC_P2_Srobovanie.AlarmTime.PT:= T#30s;
            SC_P2_Srobovanie.IdleTime.IN:= TRUE;

            IF NOT SC_P2_Srobovanie.Switch1 THEN
                P2_Srobovanie.SkrutkovaciSet_M5.Cistenie:= TRUE;
                SC_P2_Srobovanie.Switch1:= TRUE;
            END_IF

            IF P2_Srobovanie.SkrutkovaciSet_M5.CistenieUkoncene AND P2_Srobovanie.IN.SkrutkM5_ZASUNUTY_MS11 THEN
                P2_Srobovanie.SkrutkovaciSet_M5.Cistenie:= FALSE;
            END_IF

            IF NOT P2_Srobovanie.SkrutkovaciSet_M5.Cistenie AND P2_Srobovanie.SkrutkovaciSet_M5.SkrutkaM5_Pripravena AND SC_P2_Srobovanie.Switch1 THEN
                P2_Srobovanie.STAV.Cistenie_M5_BUSY:= FALSE;
                SC_P2_Srobovanie.ResetStep:= TRUE;
                SC_P2_Srobovanie.Step:= FazaNavratu;
            ELSIF SC_P2_Srobovanie.IdleTime.Q THEN
                SC_P2_Srobovanie.ResetStep:= TRUE;
                SC_P2_Srobovanie.Step:= 515;
            END_IF

        515:
            SC_P2_Srobovanie.StepName:='505 - Inicializacia - cakam na opatovne spustenie cistenia skrutkovacky M5';
            SC_P2_Srobovanie.IdleTime.PT:= T#2s;
            SC_P2_Srobovanie.AlarmTime.PT:= T#30s;

            IF NOT SC_P2_Srobovanie.Switch1 THEN
                P2_Srobovanie.SkrutkovaciSet_M5.Reset:= TRUE;
                P2_Srobovanie.SkrutkovaciSet_M5.Cistenie:= FALSE;
                SC_P2_Srobovanie.IdleTime.IN:= TRUE;
                SC_P2_Srobovanie.Switch1:= TRUE;
            END_IF

            IF SC_P2_Srobovanie.IdleTime.Q THEN
                SC_P2_Srobovanie.ResetStep:= TRUE;
                SC_P2_Srobovanie.Step:= 513;
            END_IF

            //Čistenie skrutkovačky M6//

        520:
            SC_P2_Srobovanie.StepName:='520 - Automaticky Rezim - cistenie skrutkovacky M6';
            SC_P2_Srobovanie.IdleTime.PT:= T#200ms;
            SC_P2_Srobovanie.AlarmTime.PT:= T#5s;

            P2_Srobovanie.PAR.OsX_ZadanaPozicia:= 50; //mm
            P2_Srobovanie.PAR.OsY_ZadanaPozicia:= 0; //mm

            IF NOT SC_P2_Srobovanie.Switch1 AND SC_OvlManipulatora_OsX.Step = 1 AND SC_OvlManipulatora_OsY.Step = 1 AND P2_Srobovacky_VychodziaPozicia AND Safety.STAV.P2_ZonaBunky_AKTIVNA THEN
                P2_Srobovanie.SkrutkovaciSet_M6.SkrutkaM6_Odobrata:= FALSE;
                P2_Srobovanie.SkrutkovaciSet_M6.Automat:= TRUE;
                P2_Srobovanie.SkrutkovaciSet_M6.Reset:= TRUE;
                OsX_POLOHUJ:= TRUE;
                SC_P2_Srobovanie.Switch1:= TRUE;
            END_IF

            IF NOT SC_P2_Srobovanie.Switch2 AND SC_OvlManipulatora_OsY.Step = 1 AND P2_Srobovacky_VychodziaPozicia AND P2_Srobovanie.STAV.OsX_PoziciaDosiahnuta AND Safety.STAV.P2_ZonaBunky_AKTIVNA THEN
                OsY_POLOHUJ:= TRUE;
                SC_P2_Srobovanie.Switch2:= TRUE;
            END_IF

            IF P2_Srobovanie.STAV.OsX_PoziciaDosiahnuta AND P2_Srobovanie.STAV.OsY_PoziciaDosiahnuta THEN
                P2_Srobovanie.STAV.OsX_PoziciaDosiahnuta:= FALSE;
                P2_Srobovanie.STAV.OsY_PoziciaDosiahnuta:= FALSE;
                SC_P2_Srobovanie.ResetStep:= TRUE;
                SC_P2_Srobovanie.Step:= 523;
            END_IF

        523:
            SC_P2_Srobovanie.StepName:='523 - Inicializacia - zahodenie skrutky M6';
            SC_P2_Srobovanie.IdleTime.PT:= T#30s;
            SC_P2_Srobovanie.AlarmTime.PT:= T#30s;
            SC_P2_Srobovanie.IdleTime.IN:= TRUE;

            IF NOT SC_P2_Srobovanie.Switch1 THEN
                P2_Srobovanie.SkrutkovaciSet_M6.Cistenie:= TRUE;
                SC_P2_Srobovanie.Switch1:= TRUE;
            END_IF

            IF P2_Srobovanie.SkrutkovaciSet_M6.CistenieUkoncene AND P2_Srobovanie.IN.SkrutkM6_ZASUNUTY_MS14 THEN
                P2_Srobovanie.SkrutkovaciSet_M6.Cistenie:= FALSE;
            END_IF

            IF NOT P2_Srobovanie.SkrutkovaciSet_M6.Cistenie AND P2_Srobovanie.SkrutkovaciSet_M6.SkrutkaM6_Pripravena AND SC_P2_Srobovanie.Switch1 THEN
                P2_Srobovanie.STAV.Cistenie_M6_BUSY:= FALSE;
                SC_P2_Srobovanie.ResetStep:= TRUE;
                SC_P2_Srobovanie.Step:= FazaNavratu;
            ELSIF SC_P2_Srobovanie.IdleTime.Q THEN
                SC_P2_Srobovanie.ResetStep:= TRUE;
                SC_P2_Srobovanie.Step:= 525;
            END_IF

        525:
            SC_P2_Srobovanie.StepName:='525 - Inicializacia - cakam na opatovne spustenie cistenia skrutkovacky M6';
            SC_P2_Srobovanie.IdleTime.PT:= T#2s;
            SC_P2_Srobovanie.AlarmTime.PT:= T#30s;

            IF NOT SC_P2_Srobovanie.Switch1 THEN
                P2_Srobovanie.SkrutkovaciSet_M6.Reset:= TRUE;
                P2_Srobovanie.SkrutkovaciSet_M6.Cistenie:= FALSE;
                SC_P2_Srobovanie.IdleTime.IN:= TRUE;
                SC_P2_Srobovanie.Switch1:= TRUE;
            END_IF

            IF SC_P2_Srobovanie.IdleTime.Q THEN
                SC_P2_Srobovanie.ResetStep:= TRUE;
                SC_P2_Srobovanie.Step:= 523;
            END_IF

            //*******************************************************Manuálny režim*******************************************************************************//
        700:
            SC_P2_Srobovanie.StepName:='700 - Manualny Rezim';
            SC_P2_Srobovanie.IdleTime.PT:= T#8s;
            SC_P2_Srobovanie.AlarmTime.PT:= T#5s;

            P2_Srobovanie.ServoManipulOsX_M10.PAR.JoggAcceleration:= (P2_Srobovanie.PAR.OsX_JoggRychlost * 10);
            P2_Srobovanie.ServoManipulOsX_M10.PAR.JoggDeceleration:= (P2_Srobovanie.PAR.OsX_JoggRychlost * 10);
            P2_Srobovanie.ServoManipulOsX_M10.PAR.JoggVelocity:= P2_Srobovanie.PAR.OsX_JoggRychlost;
            P2_Srobovanie.ServoManipulOsX_M10.PAR.JoggPoziciaLimitVPRED:= 60.0;
            P2_Srobovanie.ServoManipulOsX_M10.PAR.JoggPoziciaLimitVZAD:= 0.0;
            P2_Srobovanie.ServoManipulOsX_M10.CMD.JoggLimit_ACTIVE:= TRUE;

            P2_Srobovanie.ServoManipulOsY_M9.PAR.JoggAcceleration:= (P2_Srobovanie.PAR.OsY_JoggRychlost * 10);
            P2_Srobovanie.ServoManipulOsY_M9.PAR.JoggDeceleration:= (P2_Srobovanie.PAR.OsY_JoggRychlost * 10);
            P2_Srobovanie.ServoManipulOsY_M9.PAR.JoggVelocity:= P2_Srobovanie.PAR.OsY_JoggRychlost;
            P2_Srobovanie.ServoManipulOsY_M9.PAR.JoggPoziciaLimitVPRED:= 320.0;
            P2_Srobovanie.ServoManipulOsY_M9.PAR.JoggPoziciaLimitVZAD:= 0.0;
            P2_Srobovanie.ServoManipulOsY_M9.CMD.JoggLimit_ACTIVE:= TRUE;

            //Ovládanie vysunutia skrutkovačky M4//
            P2_Srobovanie.OUT.SkrutkM4_VYSUN_YV24:= P2_Srobovanie.RR_SkrutkovackuM4_VYSUN;

            //Ovládanie vysunutia skrutkovačky M5//
            P2_Srobovanie.OUT.SkrutkM5_VYSUN_YV14:= P2_Srobovanie.RR_SkrutkovackuM5_VYSUN;

            //Ovládanie vysunutia skrutkovačky M6//
            P2_Srobovanie.OUT.SkrutkM6_VYSUN_YV34:= P2_Srobovanie.RR_SkrutkovackuM6_VYSUN;

            //Spustenie čistenia skrutkovačiek//
            IF P2_Srobovanie.RR_SkrutkovackaM4_CISTENIE THEN
                P2_Srobovanie.RR_SkrutkovackaM4_CISTENIE:= FALSE;
                P2_Srobovanie.STAV.Cistenie_M4_BUSY:= TRUE;
                FazaNavratu:= 700;
                SC_P2_Srobovanie.ResetStep:= TRUE;
                SC_P2_Srobovanie.Step:= 500;
            ELSIF P2_Srobovanie.RR_SkrutkovackaM5_CISTENIE THEN
                P2_Srobovanie.RR_SkrutkovackaM5_CISTENIE:= FALSE;
                P2_Srobovanie.STAV.Cistenie_M5_BUSY:= TRUE;
                FazaNavratu:= 700;
                SC_P2_Srobovanie.ResetStep:= TRUE;
                SC_P2_Srobovanie.Step:= 510;
            ELSIF P2_Srobovanie.RR_SkrutkovackaM6_CISTENIE THEN
                P2_Srobovanie.RR_SkrutkovackaM6_CISTENIE:= FALSE;
                P2_Srobovanie.STAV.Cistenie_M6_BUSY:= TRUE;
                FazaNavratu:= 700;
                SC_P2_Srobovanie.ResetStep:= TRUE;
                SC_P2_Srobovanie.Step:= 520;
            END_IF

            //Polohovanie na pozície skrutiek//
            IF P2_Srobovanie.RR_PolohujNaPoziciuSkrutky_4F THEN
                IF P2_Srobovanie.PAR.RR_IndexPozicieSkrutky_4F = 0 THEN  //Lavá M6
                    SC_P2_Srobovanie.ResetStep:= TRUE;
                    SC_P2_Srobovanie.Step:= 110;
                ELSIF P2_Srobovanie.PAR.RR_IndexPozicieSkrutky_4F = 1 THEN  //Pravá M6
                    SC_P2_Srobovanie.ResetStep:= TRUE;
                    SC_P2_Srobovanie.Step:= 130;
                ELSIF P2_Srobovanie.PAR.RR_IndexPozicieSkrutky_4F = 2 THEN  //Lavá M4
                    SC_P2_Srobovanie.ResetStep:= TRUE;
                    SC_P2_Srobovanie.Step:= 150;
                ELSIF P2_Srobovanie.PAR.RR_IndexPozicieSkrutky_4F = 3 THEN  //Pravá M4
                    SC_P2_Srobovanie.ResetStep:= TRUE;
                    SC_P2_Srobovanie.Step:= 170;
                END_IF
            ELSIF P2_Srobovanie.RR_PolohujNaPoziciuSkrutky_5F THEN
                IF P2_Srobovanie.PAR.RR_IndexPozicieSkrutky_5F = 0 THEN  //Lavá M6
                    SC_P2_Srobovanie.ResetStep:= TRUE;
                    SC_P2_Srobovanie.Step:= 200;
                ELSIF P2_Srobovanie.PAR.RR_IndexPozicieSkrutky_5F = 1 THEN  //Pravá M6
                    SC_P2_Srobovanie.ResetStep:= TRUE;
                    SC_P2_Srobovanie.Step:= 220;
                ELSIF P2_Srobovanie.PAR.RR_IndexPozicieSkrutky_5F = 2 THEN  //Lavá M4
                    SC_P2_Srobovanie.ResetStep:= TRUE;
                    SC_P2_Srobovanie.Step:= 240;
                ELSIF P2_Srobovanie.PAR.RR_IndexPozicieSkrutky_5F = 3 THEN  //Pravá M4
                    SC_P2_Srobovanie.ResetStep:= TRUE;
                    SC_P2_Srobovanie.Step:= 260;
                END_IF
            ELSIF  P2_Srobovanie.RR_PolohujNaPoziciuSkrutky_5H THEN
                IF P2_Srobovanie.PAR.RR_IndexPozicieSkrutky_5H = 0 THEN  //Lavá M5
                    SC_P2_Srobovanie.ResetStep:= TRUE;
                    SC_P2_Srobovanie.Step:= 300;
                ELSIF P2_Srobovanie.PAR.RR_IndexPozicieSkrutky_5H = 1 THEN  //Pravá M5
                    SC_P2_Srobovanie.ResetStep:= TRUE;
                    SC_P2_Srobovanie.Step:= 320;
                ELSIF P2_Srobovanie.PAR.RR_IndexPozicieSkrutky_5H = 2 THEN  //Stredná M4
                    SC_P2_Srobovanie.ResetStep:= TRUE;
                    SC_P2_Srobovanie.Step:= 340;
                END_IF
            END_IF

    END_CASE

            END_PROGRAM

PROGRAM _EXIT
            (* Insert code here *)

            END_PROGRAM
```

#### Variables.var - Local variables
```iecst
VAR
	SC_OvlManipulatora_OsX : SequenceControlTyp;
	OsX_JoggVPRED : BOOL;
	OsX_JoggVZAD : BOOL;
	OsX_POLOHUJ : BOOL;
	OsX_HOME : BOOL;
	OsX_STOP : BOOL;
	SC_OvlManipulatora_OsY : SequenceControlTyp;
	OsY_JoggVPRED : BOOL;
	OsY_JoggVZAD : BOOL;
	OsY_POLOHUJ : BOOL;
	OsY_HOME : BOOL;
	OsY_STOP : BOOL;
	Test : BOOL;
	ZadanaPoziciaUINT_OsX : UINT;
	AktualnaPoziciaUINT_OsX : UINT;
	ZadanaPoziciaUINT_OsY : UINT;
	AktualnaPoziciaUINT_OsY : UINT;
	Triger_0 : BOOL;
	TEST : BOOL;
	CasPowerON_OsX : TON;
	CasPowerON_OsY : TON;
	PAUZA : BOOL;
	i : USINT;
	CasSrobovania : REAL;
	M5_DosiahnutyMoment_REAL : REAL;
	M5_Moment_ToleranciaMAX_REAL : REAL;
	M5_Moment_ToleranciaMIN_REAL : REAL;
	M4_DosiahnutyMoment_REAL : REAL;
	M4_Moment_ToleranciaMAX_REAL : REAL;
	M4_Moment_ToleranciaMIN_REAL : REAL;
	M6_DosiahnutyMoment_REAL : REAL;
	M6_Moment_ToleranciaMAX_REAL : REAL;
	M6_Moment_ToleranciaMIN_REAL : REAL;
	M5_PrevodMomentu : PrevodMomentu;
	M6_PrevodMomentu : PrevodMomentu;
	M4_PrevodMomentu : PrevodMomentu;
	CasZastaveniaServa : TON;
	CasZastaveniaServa_2 : TON;
	FazaNavratu : UINT;
	CasKontrolyZasobSkrutiek_M4 : TON;
	CasKontrolyZasobSkrutiek_M5 : TON;
	CasKontrolyZasobSkrutiek_M6 : TON;
END_VAR
(******Zápis do ParID serva*************)
VAR
	MC_BR_ProcessParID_AcpAx_0 : MC_BR_ProcessParID_AcpAx := (0);
	McAcpAxProcessParIDType_0 : ARRAY[0..1] OF McAcpAxProcessParIDType;
	OsX_NovaHodnotaMomentu_POS : REAL := 0.0;
	OsX_NovaHodnotaMomentu_NEG : REAL := 0.0;
	MC_BR_ProcessParID_AcpAx_1 : MC_BR_ProcessParID_AcpAx := (0);
	McAcpAxProcessParIDType_1 : ARRAY[0..1] OF McAcpAxProcessParIDType;
	OsY_NovaHodnotaMomentu_POS : REAL := 0.0;
	OsY_NovaHodnotaMomentu_NEG : REAL := 0.0;
END_VAR
```

#### OvlManipulatora_OsX.st
```iecst
ACTION OvlManipulatora_OsX:

	//*****************************Axis 3************************************//
	//Otáčka serva = 10mm//
	//Motor má absolútny encodér//

    //ENABLE knižnice//
    IF P2_Srobovanie.ServoManipulOsX_M10.STATUS.Communication_READY THEN
        P2_Srobovanie.ServoManipulOsX_M10.CMD.ENABLE:= TRUE;
    ELSE
        P2_Srobovanie.ServoManipulOsX_M10.CMD.ENABLE:= FALSE;
    END_IF

	//Zapnutie serva//
	CasPowerON_OsX.IN:= P2_Srobovanie.ServoManipulOsX_M10.STATUS.ReadyToPower_ON AND P2_Srobovanie.STAV.OsX_LimitSnimace_BUSY AND P2_Srobovanie.ServoManipulOsX_M10.STATUS.EnableSwitch_ACTIVE AND NOT P2_Srobovanie.ServoManipulOsX_M10.STATUS.ERROR;
	IF CasPowerON_OsX.Q THEN
		P2_Srobovanie.ServoManipulOsX_M10.CMD.POWER:= TRUE;
	ELSE
		P2_Srobovanie.ServoManipulOsX_M10.CMD.POWER:= FALSE;
	END_IF

	CasPowerON_OsX.PT:= T#1s;
	CasPowerON_OsX();

    //Zobrazenie stavou a parametrov serva//
    P2_Srobovanie.STAV.OsX_AktualnaPozicia:= P2_Srobovanie.ServoManipulOsX_M10.STATUS.ActualPosition;
    P2_Srobovanie.STAV.OsX_AktualnaRychlost:= P2_Srobovanie.ServoManipulOsX_M10.STATUS.ActualVelocity;
	P2_Srobovanie.STAV.OsX_AktualnyMoment:= P2_Srobovanie.ServoManipulOsX_M10.STATUS.ActualTorque;
	P2_Srobovanie.STAV.OsX_HomingOK:= P2_Srobovanie.ServoManipulOsX_M10.STATUS.Homing_OK;
	P2_Srobovanie.STAV.OsX_BUSY:= P2_Srobovanie.ServoManipulOsX_M10.STATUS.MoveAbsolute_BUSY;
	P2_Srobovanie.STAV.OsX_JoggLimitDosiahnuty:= P2_Srobovanie.ServoManipulOsX_M10.STATUS.JoggLimit_Dosiahnuty;

	//Zadané parametre serva//
	P2_Srobovanie.ServoManipulOsX_M10.HomePAR.Acceleration:= 50;
	P2_Srobovanie.ServoManipulOsX_M10.HomePAR.HomingVelocity:= 2;
	P2_Srobovanie.ServoManipulOsX_M10.HomePAR.StartVelocity:= 5;
	P2_Srobovanie.ServoManipulOsX_M10.HomePAR.Position:= -21653.3;    //Offset homing pozície pre absolutny snímač
	P2_Srobovanie.ServoManipulOsX_M10.HomePAR.HomingMode:= 3; //0 - direct, 1- refrenčný snímač, 2 - limitný snímač, 3 - absolutny encoder, 4 - na moment//

	P2_Srobovanie.ServoManipulOsX_M10.PAR.Acceleration:= P2_RemPremenne.P2_ManipSrob_OsX_Rychlost*10;
	P2_Srobovanie.ServoManipulOsX_M10.PAR.Deceleration:= P2_RemPremenne.P2_ManipSrob_OsX_Rychlost*10;
	P2_Srobovanie.ServoManipulOsX_M10.PAR.StopDeceleration:= P2_RemPremenne.P2_ManipSrob_OsX_Rychlost*10;
	P2_Srobovanie.ServoManipulOsX_M10.PAR.Velocity:= P2_RemPremenne.P2_ManipSrob_OsX_Rychlost;
	P2_Srobovanie.ServoManipulOsX_M10.PAR.Position:= P2_Srobovanie.PAR.OsX_ZadanaPozicia;

	//Zastavenie pohybu serva//
	IF OsX_STOP THEN
		P2_Srobovanie.ServoManipulOsX_M10.CMD.STOP:= TRUE;
		SC_OvlManipulatora_OsX.Step:= 0;
		CasZastaveniaServa.IN:= TRUE;
		OsX_STOP:= FALSE;
	END_IF

	IF CasZastaveniaServa.Q THEN
		P2_Srobovanie.ServoManipulOsX_M10.CMD.STOP:= FALSE;
		CasZastaveniaServa.IN:= FALSE;
	END_IF

	CasZastaveniaServa.PT:= T#2s;
	CasZastaveniaServa();

	//Volanie funkcie SequenceControl//
	SequenceControl(SC:= SC_OvlManipulatora_OsX);

	CASE SC_OvlManipulatora_OsX.Step OF

		0:
			SC_OvlManipulatora_OsX.StepName:= '0 - Nulovanie';
			OsX_JoggVPRED:= FALSE;
			OsX_JoggVZAD:= FALSE;
			OsX_POLOHUJ:= FALSE;
			OsX_HOME:= FALSE;
			P2_Srobovanie.ServoManipulOsX_M10.CMD.HOME:= FALSE;
			P2_Srobovanie.ServoManipulOsX_M10.CMD.JoggVPRED:= FALSE;
			P2_Srobovanie.ServoManipulOsX_M10.CMD.JoggVZAD:= FALSE;
			P2_Srobovanie.ServoManipulOsX_M10.CMD.MoveAbsolute:= FALSE;

			IF SC_P2_Srobovanie.Step <> 0 AND P2_Srobovanie.ServoManipulOsX_M10.STATUS.Power_ON AND NOT P2_Srobovanie.ServoManipulOsX_M10.STATUS.ERROR AND NOT P2_Srobovanie.ServoManipulOsX_M10.STATUS.STOP_ACTIVE THEN
				SC_OvlManipulatora_OsX.ResetStep:= TRUE;
				SC_OvlManipulatora_OsX.Step:= 1;
			END_IF

		1:
			SC_OvlManipulatora_OsX.StepName:= '1 - Rozhodnutie o cinnosti';
			IF OsX_JoggVPRED THEN
				SC_OvlManipulatora_OsX.Step:= 10;
			ELSIF OsX_JoggVZAD THEN
				SC_OvlManipulatora_OsX.Step:= 20;
			ELSIF OsX_HOME THEN
				SC_OvlManipulatora_OsX.Step:= 30;
			ELSIF OsX_POLOHUJ THEN
				SC_OvlManipulatora_OsX.Step:= 40;
			END_IF

		10:
			SC_OvlManipulatora_OsX.StepName:= '10 - Jogg VPRED';
			SC_OvlManipulatora_OsX.IdleTime.PT:= T#3s;
			SC_OvlManipulatora_OsX.AlarmTime.PT:= T#3s;

			IF NOT SC_OvlManipulatora_OsX.Switch1 THEN
				P2_Srobovanie.ServoManipulOsX_M10.CMD.JoggVPRED:= TRUE;
				SC_OvlManipulatora_OsX.Switch1:= TRUE;
			END_IF

			IF NOT OsX_JoggVPRED THEN
				SC_OvlManipulatora_OsX.ResetStep:= TRUE;
				SC_OvlManipulatora_OsX.Step:= 0;
			END_IF

		20:
			SC_OvlManipulatora_OsX.StepName:= '20 - Jogg VZAD';
			SC_OvlManipulatora_OsX.IdleTime.PT:= T#3s;
			SC_OvlManipulatora_OsX.AlarmTime.PT:= T#3s;

			IF NOT SC_OvlManipulatora_OsX.Switch1 THEN
				P2_Srobovanie.ServoManipulOsX_M10.CMD.JoggVZAD:= TRUE;
				SC_OvlManipulatora_OsX.Switch1:= TRUE;
			END_IF

			IF NOT OsX_JoggVZAD THEN
				SC_OvlManipulatora_OsX.ResetStep:= TRUE;
				SC_OvlManipulatora_OsX.Step:= 0;
			END_IF

		30:
			SC_OvlManipulatora_OsX.StepName:= '30 - Homing';
			SC_OvlManipulatora_OsX.IdleTime.PT:= T#500ms;
			SC_OvlManipulatora_OsX.AlarmTime.PT:= T#3s;

			IF NOT SC_OvlManipulatora_OsX.Switch1 THEN
				P2_Srobovanie.ServoManipulOsX_M10.CMD.HOME:= TRUE;
				SC_OvlManipulatora_OsX.IdleTime.IN:= TRUE;
				SC_OvlManipulatora_OsX.Switch1:= TRUE;
			END_IF

			IF P2_Srobovanie.ServoManipulOsX_M10.STATUS.Homing_OK AND SC_OvlManipulatora_OsX.IdleTime.Q THEN
				SC_OvlManipulatora_OsX.ResetStep:= TRUE;
				SC_OvlManipulatora_OsX.Step:= 0;
			END_IF

		40:
			SC_OvlManipulatora_OsX.StepName:= '40 - Polohovanie';
			SC_OvlManipulatora_OsX.IdleTime.PT:= T#500ms;
			SC_OvlManipulatora_OsX.AlarmTime.PT:= T#3s;

			ZadanaPoziciaUINT_OsX:= LREAL_TO_UINT(P2_Srobovanie.PAR.OsX_ZadanaPozicia);
			AktualnaPoziciaUINT_OsX:= LREAL_TO_UINT(P2_Srobovanie.STAV.OsX_AktualnaPozicia);

			IF NOT SC_OvlManipulatora_OsX.Switch1 THEN
				P2_Srobovanie.ServoManipulOsX_M10.CMD.MoveAbsolute:= TRUE;
				SC_OvlManipulatora_OsX.Switch1:= TRUE;
			END_IF

			IF (AktualnaPoziciaUINT_OsX = ZadanaPoziciaUINT_OsX) AND P2_Srobovanie.ServoManipulOsX_M10.STATUS.MoveAbsolute_DONE THEN
				P2_Srobovanie.STAV.OsX_PoziciaDosiahnuta:= TRUE;
				SC_OvlManipulatora_OsX.ResetStep:= TRUE;
				SC_OvlManipulatora_OsX.Step:= 0;
			END_IF

	END_CASE

END_ACTION
```

#### OvlManipulatora_OsY.st
```iecst
ACTION OvlManipulatora_OsY:

	//************************Axis 4*******************************//
	//Otáčka serva = 10mm//
	//Motor má absolútny encodér//

    //ENABLE knižnice//
    IF P2_Srobovanie.ServoManipulOsY_M9.STATUS.Communication_READY THEN
        P2_Srobovanie.ServoManipulOsY_M9.CMD.ENABLE:= TRUE;
    ELSE
        P2_Srobovanie.ServoManipulOsY_M9.CMD.ENABLE:= FALSE;
    END_IF

	//Zapnutie serva//
	CasPowerON_OsY.IN:= P2_Srobovanie.ServoManipulOsY_M9.STATUS.ReadyToPower_ON AND P2_Srobovanie.STAV.OsY_LimitSnimace_BUSY AND P2_Srobovanie.ServoManipulOsY_M9.STATUS.EnableSwitch_ACTIVE AND NOT P2_Srobovanie.ServoManipulOsY_M9.STATUS.ERROR;
	IF CasPowerON_OsY.Q THEN
		P2_Srobovanie.ServoManipulOsY_M9.CMD.POWER:= TRUE;
	ELSE
		P2_Srobovanie.ServoManipulOsY_M9.CMD.POWER:= FALSE;
	END_IF

	CasPowerON_OsY.PT:= T#1s;
	CasPowerON_OsY();

    //Zobrazenie stavou a parametrov serva//
    P2_Srobovanie.STAV.OsY_AktualnaPozicia:= P2_Srobovanie.ServoManipulOsY_M9.STATUS.ActualPosition;
    P2_Srobovanie.STAV.OsY_AktualnaRychlost:= P2_Srobovanie.ServoManipulOsY_M9.STATUS.ActualVelocity;
	P2_Srobovanie.STAV.OsY_AktualnyMoment:= P2_Srobovanie.ServoManipulOsY_M9.STATUS.ActualTorque;
	P2_Srobovanie.STAV.OsY_HomingOK:= P2_Srobovanie.ServoManipulOsY_M9.STATUS.Homing_OK;
	P2_Srobovanie.STAV.OsY_BUSY:= P2_Srobovanie.ServoManipulOsY_M9.STATUS.MoveAbsolute_BUSY;
	P2_Srobovanie.STAV.OsY_JoggLimitDosiahnuty:= P2_Srobovanie.ServoManipulOsY_M9.STATUS.JoggLimit_Dosiahnuty;

	//Zadané parametre serva//
	P2_Srobovanie.ServoManipulOsY_M9.HomePAR.Acceleration:= 50;
	P2_Srobovanie.ServoManipulOsY_M9.HomePAR.HomingVelocity:= 2;
	P2_Srobovanie.ServoManipulOsY_M9.HomePAR.StartVelocity:= 5;
	P2_Srobovanie.ServoManipulOsY_M9.HomePAR.Position:= -22260.4;    //Offset homing pozície pre absolutny snímač
	P2_Srobovanie.ServoManipulOsY_M9.HomePAR.HomingMode:= 3; //0 - direct, 1- refrenčný snímač, 2 - limitný snímač, 3 - absolutny encoder, 4 - na moment//

	P2_Srobovanie.ServoManipulOsY_M9.PAR.Acceleration:= P2_RemPremenne.P2_ManipSrob_OsY_Rychlost*10;
	P2_Srobovanie.ServoManipulOsY_M9.PAR.Deceleration:= P2_RemPremenne.P2_ManipSrob_OsY_Rychlost*10;
	P2_Srobovanie.ServoManipulOsY_M9.PAR.StopDeceleration:= P2_RemPremenne.P2_ManipSrob_OsY_Rychlost*10;
	P2_Srobovanie.ServoManipulOsY_M9.PAR.Velocity:= P2_RemPremenne.P2_ManipSrob_OsY_Rychlost;
	P2_Srobovanie.ServoManipulOsY_M9.PAR.Position:= P2_Srobovanie.PAR.OsY_ZadanaPozicia;

	//Zastavenie pohybu serva//
	IF OsY_STOP THEN
		P2_Srobovanie.ServoManipulOsY_M9.CMD.STOP:= TRUE;
		SC_OvlManipulatora_OsY.Step:= 0;
		CasZastaveniaServa_2.IN:= TRUE;
		OsY_STOP:= FALSE;
	END_IF

	IF CasZastaveniaServa_2.Q THEN
		P2_Srobovanie.ServoManipulOsY_M9.CMD.STOP:= FALSE;
		CasZastaveniaServa_2.IN:= FALSE;
	END_IF

	CasZastaveniaServa_2.PT:= T#2s;
	CasZastaveniaServa_2();

	//Volanie funkcie SequenceControl//
	SequenceControl(SC:= SC_OvlManipulatora_OsY);

	CASE SC_OvlManipulatora_OsY.Step OF

		0:
			SC_OvlManipulatora_OsY.StepName:= '0 - Nulovanie';
			OsY_JoggVPRED:= FALSE;
			OsY_JoggVZAD:= FALSE;
			OsY_POLOHUJ:= FALSE;
			OsY_HOME:= FALSE;
			P2_Srobovanie.ServoManipulOsY_M9.CMD.HOME:= FALSE;
			P2_Srobovanie.ServoManipulOsY_M9.CMD.JoggVPRED:= FALSE;
			P2_Srobovanie.ServoManipulOsY_M9.CMD.JoggVZAD:= FALSE;
			P2_Srobovanie.ServoManipulOsY_M9.CMD.MoveAbsolute:= FALSE;

			IF SC_P2_Srobovanie.Step <> 0 AND P2_Srobovanie.ServoManipulOsY_M9.STATUS.Power_ON AND NOT P2_Srobovanie.ServoManipulOsY_M9.STATUS.ERROR AND NOT P2_Srobovanie.ServoManipulOsY_M9.STATUS.STOP_ACTIVE THEN
				SC_OvlManipulatora_OsY.ResetStep:= TRUE;
				SC_OvlManipulatora_OsY.Step:= 1;
			END_IF

		1:
			SC_OvlManipulatora_OsY.StepName:= '1 - Rozhodnutie o cinnosti';
			IF OsY_JoggVPRED THEN
				SC_OvlManipulatora_OsY.Step:= 10;
			ELSIF OsY_JoggVZAD THEN
				SC_OvlManipulatora_OsY.Step:= 20;
			ELSIF OsY_HOME THEN
				SC_OvlManipulatora_OsY.Step:= 30;
			ELSIF OsY_POLOHUJ THEN
				SC_OvlManipulatora_OsY.Step:= 40;
			END_IF

		10:
			SC_OvlManipulatora_OsY.StepName:= '10 - Jogg VPRED';
			SC_OvlManipulatora_OsY.IdleTime.PT:= T#3s;
			SC_OvlManipulatora_OsY.AlarmTime.PT:= T#3s;

			IF NOT SC_OvlManipulatora_OsY.Switch1 THEN
				P2_Srobovanie.ServoManipulOsY_M9.CMD.JoggVPRED:= TRUE;
				SC_OvlManipulatora_OsY.Switch1:= TRUE;
			END_IF

			IF NOT OsY_JoggVPRED THEN
				SC_OvlManipulatora_OsY.ResetStep:= TRUE;
				SC_OvlManipulatora_OsY.Step:= 0;
			END_IF

		20:
			SC_OvlManipulatora_OsY.StepName:= '20 - Jogg VZAD';
			SC_OvlManipulatora_OsY.IdleTime.PT:= T#3s;
			SC_OvlManipulatora_OsY.AlarmTime.PT:= T#3s;

			IF NOT SC_OvlManipulatora_OsY.Switch1 THEN
				P2_Srobovanie.ServoManipulOsY_M9.CMD.JoggVZAD:= TRUE;
				SC_OvlManipulatora_OsY.Switch1:= TRUE;
			END_IF

			IF NOT OsY_JoggVZAD THEN
				SC_OvlManipulatora_OsY.ResetStep:= TRUE;
				SC_OvlManipulatora_OsY.Step:= 0;
			END_IF

		30:
			SC_OvlManipulatora_OsY.StepName:= '30 - Homing';
			SC_OvlManipulatora_OsY.IdleTime.PT:= T#500ms;
			SC_OvlManipulatora_OsY.AlarmTime.PT:= T#3s;

			IF NOT SC_OvlManipulatora_OsY.Switch1 THEN
				P2_Srobovanie.ServoManipulOsY_M9.CMD.HOME:= TRUE;
				SC_OvlManipulatora_OsY.IdleTime.IN:= TRUE;
				SC_OvlManipulatora_OsY.Switch1:= TRUE;
			END_IF

			IF P2_Srobovanie.ServoManipulOsY_M9.STATUS.Homing_OK AND SC_OvlManipulatora_OsY.IdleTime.Q THEN
				SC_OvlManipulatora_OsY.ResetStep:= TRUE;
				SC_OvlManipulatora_OsY.Step:= 0;
			END_IF

		40:
			SC_OvlManipulatora_OsY.StepName:= '40 - Polohovanie';
			SC_OvlManipulatora_OsY.IdleTime.PT:= T#500ms;
			SC_OvlManipulatora_OsY.AlarmTime.PT:= T#3s;

			ZadanaPoziciaUINT_OsY:= LREAL_TO_UINT(P2_Srobovanie.PAR.OsY_ZadanaPozicia);
			AktualnaPoziciaUINT_OsY:= LREAL_TO_UINT(P2_Srobovanie.STAV.OsY_AktualnaPozicia);

			IF NOT SC_OvlManipulatora_OsY.Switch1 THEN
				P2_Srobovanie.ServoManipulOsY_M9.CMD.MoveAbsolute:= TRUE;
				SC_OvlManipulatora_OsY.Switch1:= TRUE;
			END_IF

			IF (AktualnaPoziciaUINT_OsY = ZadanaPoziciaUINT_OsY) AND P2_Srobovanie.ServoManipulOsY_M9.STATUS.MoveAbsolute_DONE THEN
				P2_Srobovanie.STAV.OsY_PoziciaDosiahnuta:= TRUE;
				SC_OvlManipulatora_OsY.ResetStep:= TRUE;
				SC_OvlManipulatora_OsY.Step:= 0;
			END_IF

	END_CASE

END_ACTION
```
